// TIA Portal V16 export
// export: Created 2022-02-28T20:45:46.1810746Z, ExportSetting WithDefaults, DisplayName Totally Integrated Automation Portal, DisplayVersion V16, DisplayName TIA Portal Version Control Interface, DisplayVersion V16, DisplayName TIA Portal Openness, DisplayVersion V16, DisplayName STEP 7 Professional, DisplayVersion V16, DisplayName STEP 7 Safety, DisplayVersion V16, DisplayName WinCC Advanced, DisplayVersion V16
DATA_BLOCK "04_Cam_Pentoflex"   // DB4
{ S7_Optimized_Access := 'TRUE' }
VERSION : 0.1
// stored: AutoNumber true, DBAccessibleFromOPCUA true, IsOnlyStoredInLoadMemory false, IsRetainMemResEnabled false, IsWriteProtectedInAS false, MemoryReserve 100
   VAR
      Trigger_Enable_Cam2 : Bool;   // 1= Disparador Ethernet Habilitado
      Trigger : Bool;   // Adquirir imagen
      Status_Register : Array[0..7] of Bool;
      BufferResultsEnable : Bool;
      DecodeStatusRegister : Array[0..7] of Bool;
      ResultsAck : Bool;
      DecodeResult : Struct
         ResultsID : UInt;
         ResultCode : UInt;
         ResultExtended : UInt;
         ResultLength : UInt;
         ResultData : Array[0..63] of Byte;   // Resultados de la ultima decodi
      END_STRUCT;
      SoftEvents : Byte;
      TriggerID : UInt;
      UserDataOption : UInt;
      UserDataLength : UInt;
      SoftEventAck : Byte;
   END_VAR
BEGIN
   Status_Register[0] := true;   // Trigger Ready
   // Status_Register[1] : Trigger Ack
   // Status_Register[2] : Reserved
   // Status_Register[3] : Missed Acquisition
   // Status_Register[4] : Reserved
   // Status_Register[5] : Reserved
   // Status_Register[6] : Reserved
   // Status_Register[7] : Reserved
   // DecodeStatusRegister[0] : Decoding
   // DecodeStatusRegister[1] : Decode Complete
   // DecodeStatusRegister[2] : Result Buffer Overrun
   // DecodeStatusRegister[3] : Result available
   // DecodeStatusRegister[4] : Reserved
   // DecodeStatusRegister[5] : Reserved
   // DecodeStatusRegister[6] : Reserved
   // DecodeStatusRegister[7] : General Fault
END_DATA_BLOCK
